// TIA Portal V20 export
DATA_BLOCK "instGetMotorstarterSignals"   // DB67
// stored: InstanceOfName GetMotorstarterSignals, InstanceOfType FB
"GetMotorstarterSignals"
   // VAR_INPUT
   //    Et200SpMotorstarterInterfaceAllUnits { ExternalAccessible := 'False'; ExternalVisible := 'False'; ExternalWritable := 'False'} : Array[1.."NO_OF_UNITS"] of "typeEmMotorStarterInterface";
   //    numberOfMS : USInt;
   // END_VAR
   // VAR_OUTPUT
   //    selectedUnit : USInt;
   //    selectedEM : USInt;
   //    error : Word;
   // END_VAR
   // VAR_IN_OUT
   //    Et200SpMotorstarterInterfaceHmi : "typeEt200SpMotorstarterInterfaceHmi";
   // END_VAR
   // VAR
   //    statSelectedEMMotorStarter : USInt;
   //    statSelectedUnitMotorStarter : USInt;
   // END_VAR
BEGIN
END_DATA_BLOCK
